(* IEC 61131-3 sources: volt/packages/volt-lsp-iec/test-corpus/bakon-nano/Device/Plc Logic/Application/Library Manager/VisuUtils, 38 files *)

(* ---- CLOSEDIALOGDATA.dut ---- *)
TYPE CLOSEDIALOGDATA :
STRUCT
	DLGMANAGER : VisuElemBase.IDialogManager;
	VISUDIALOG : VisuElemBase.IVisualisationDialog;
	DIALOGRESULT : VisuElemBase.Visu_DialogResult;
END_STRUCT
END_TYPE

(* ---- ERROR.dut ---- *)
TYPE ERROR :
(
	NO_ERROR,
	TIME_OUT,
	NOT_CALLED_FROM_VISU,
	NOT_SUPPORTED_FOR_INTEGRATED_VISU,
	ERROR,
	TRANSFER_CANCELLED,
	TRANSER_IN_PROGRESS,
	TRANSFER_FAILED,
	FILE_READ_ERROR,
	VISU_NOT_FOUND,
	NO_CLIENT_FILTER,
	NO_ITERATION_CALLBACK,
	FILE_TRANSFER_SERVICES_NOT_SUPPORTED,
	BLOCKED_DUE_TO_ONLINECHANGE,
	CANCELLED_DUE_TO_ONLINE_CHANGE
);
END_TYPE

(* ---- OPENDIALOGDATA.dut ---- *)
TYPE OPENDIALOGDATA :
STRUCT
	DLGMANAGER : VisuElemBase.IDialogManager;
	VISUDIALOG : VisuElemBase.IVisualisationDialog;
	POSITIONRECT : VisuElemBase.VisuStructSimpleRectangle;
END_STRUCT
END_TYPE

(* ---- VISUINPUTTYPE.dut ---- *)
TYPE VISUINPUTTYPE :
(
	KEYBOARD := 0,
	TOUCHSCREEN := 1
);
END_TYPE

(* ---- GLOBALS.gvl ---- *)
VAR_GLOBAL
	ALLCLIENTS : FBAcceptsAllClients;
	CURRENTCLIENT : FBAcceptsCurrentClient;
	ONLYTARGETVISU : FBAcceptsTargetVisuOnly;
	ONLYREMOTETARGETVISU : FBAcceptsRemoteTargetVisuOnly;
	ONLYWEBVISU : FBAcceptsWebVisuOnly;
END_VAR

(* ---- PUBLICVARIABLES.gvl ---- *)
VAR_GLOBAL
	CLIENTS : FbCurrentClientProvider;
END_VAR

(* ---- VARIABLES.gvl ---- *)
VAR_GLOBAL
	G_ACTIONHANDLER_INST : FbActionHandler;
	G_OCDETECTOR : FBOCStateDetector;
END_VAR

(* ---- ICAPTURECURRENTCLIENT.itf ---- *)
INTERFACE ICAPTURECURRENTCLIENT
END_INTERFACE

(* ---- IEXECUTEACTION.itf ---- *)
INTERFACE IEXECUTEACTION
END_INTERFACE

METHOD STARTEXECUTE
END_METHOD

(* ---- IVISUALIZATIONCLIENT.itf ---- *)
INTERFACE IVISUALIZATIONCLIENT
END_INTERFACE

METHOD GETCLIENTNAME : STRING
VAR_OUTPUT
	XISVALID : BOOL;
END_VAR
END_METHOD

METHOD GETIPV4ADDRESS : STRING
VAR_OUTPUT
	XISVALID : BOOL;
END_VAR
END_METHOD

METHOD GETREMOTETARGETVISUID : DWORD
VAR_OUTPUT
	XISVALID : BOOL;
END_VAR
END_METHOD

METHOD GETREMOTETARGETVISUVERSION : VERSION
VAR_OUTPUT
	XISVALID : BOOL;
END_VAR
END_METHOD

(* ---- IVISUALIZATIONCLIENTFILTER.itf ---- *)
INTERFACE IVISUALIZATIONCLIENTFILTER
END_INTERFACE

METHOD ISACCEPTED : BOOL
VAR_INPUT
	ITFCLIENT : IVisualizationClient;
END_VAR
END_METHOD

(* ---- IVISUALIZATIONCLIENTITERATION.itf ---- *)
INTERFACE IVISUALIZATIONCLIENTITERATION
END_INTERFACE

METHOD ENDITERATION
END_METHOD

METHOD HANDLECLIENT
VAR_INPUT
	ITFCLIENT : IVisualizationClient;
END_VAR
END_METHOD

METHOD STARTITERATION
END_METHOD

(* ---- IVISUALIZATIONCLIENTRAW.itf ---- *)
INTERFACE IVISUALIZATIONCLIENTRAW
END_INTERFACE

(* ---- FCTGETNEXTVISU.pou ---- *)
FUNCTION FCTGETNEXTVISU : IVisualisation
VAR_INPUT
	PCLIENT : POINTER TO VisuStructClientData;
END_VAR
END_FUNCTION

(* ---- FCTGETPREVIOUSVISU.pou ---- *)
FUNCTION FCTGETPREVIOUSVISU : IVisualisation
VAR_INPUT
	PCLIENT : POINTER TO VisuStructClientData;
END_VAR
END_FUNCTION

(* ---- GETCLIENTTAGIPV4.pou ---- *)
FUNCTION GETCLIENTTAGIPV4 : BOOL
VAR_INPUT
	PCLIENTDATA : POINTER TO VisuStructClientData;
END_VAR
VAR_IN_OUT
	SIPV4 : STRING;
END_VAR
END_FUNCTION

(* ---- GETCLIENTTAGNAME.pou ---- *)
FUNCTION GETCLIENTTAGNAME : BOOL
VAR_INPUT
	PCLIENTDATA : POINTER TO VisuStructClientData;
END_VAR
VAR_IN_OUT
	SNAME : STRING;
END_VAR
END_FUNCTION

(* ---- GETCLIENTTAGREMOTETARGETVISUID.pou ---- *)
FUNCTION GETCLIENTTAGREMOTETARGETVISUID : BOOL
VAR_INPUT
	PCLIENTDATA : POINTER TO VisuStructClientData;
END_VAR
VAR_OUTPUT
	DWID : DWORD;
END_VAR
END_FUNCTION

(* ---- GETCLIENTTAGREMOTETARGETVISUVERSION.pou ---- *)
FUNCTION GETCLIENTTAGREMOTETARGETVISUVERSION : BOOL
VAR_INPUT
	PCLIENTDATA : POINTER TO VisuStructClientData;
END_VAR
VAR_IN_OUT
	V : VERSION;
END_VAR
END_FUNCTION

(* ---- ISVISUTASK.pou ---- *)
FUNCTION ISVISUTASK : BOOL
END_FUNCTION

(* ---- FBACCEPTSALLCLIENTS.pou ---- *)
FUNCTION_BLOCK FBACCEPTSALLCLIENTS
END_FUNCTION_BLOCK

METHOD ISACCEPTED : BOOL
VAR_INPUT
	ITFCLIENT : IVisualizationClient;
END_VAR
END_METHOD

(* ---- FBACCEPTSCLIENTBYTYPEBASE.pou ---- *)
FUNCTION_BLOCK FBACCEPTSCLIENTBYTYPEBASE
VAR
	ABSTRACCEPTEDCLIENTTYPE : VisuClientType;
END_VAR
END_FUNCTION_BLOCK

METHOD ISACCEPTED : BOOL
VAR_INPUT
	ITFCLIENT : IVisualizationClient;
END_VAR
END_METHOD

(* ---- FBACCEPTSCURRENTCLIENT.pou ---- *)
FUNCTION_BLOCK FBACCEPTSCURRENTCLIENT
END_FUNCTION_BLOCK

METHOD ISACCEPTED : BOOL
VAR_INPUT
	ITFCLIENT : IVisualizationClient;
END_VAR
END_METHOD

METHOD SETCLIENT
VAR_INPUT
	PCLIENTDATA : POINTER TO VisuElemBase.VisuStructClientData;
END_VAR
END_METHOD

(* ---- FBACCEPTSREMOTETARGETVISUONLY.pou ---- *)
FUNCTION_BLOCK FBACCEPTSREMOTETARGETVISUONLY EXTENDS FBAcceptsClientByTypeBase
VAR
	ABSTRACCEPTEDCLIENTTYPE : VisuClientType;
END_VAR
END_FUNCTION_BLOCK

(* ---- FBACCEPTSTARGETVISUONLY.pou ---- *)
FUNCTION_BLOCK FBACCEPTSTARGETVISUONLY EXTENDS FBAcceptsClientByTypeBase
VAR
	ABSTRACCEPTEDCLIENTTYPE : VisuClientType;
END_VAR
END_FUNCTION_BLOCK

(* ---- FBACCEPTSWEBVISUONLY.pou ---- *)
FUNCTION_BLOCK FBACCEPTSWEBVISUONLY EXTENDS FBAcceptsClientByTypeBase
VAR
	ABSTRACCEPTEDCLIENTTYPE : VisuClientType;
END_VAR
END_FUNCTION_BLOCK

(* ---- FBACTIONHANDLER.pou ---- *)
FUNCTION_BLOCK FBACTIONHANDLER
VAR
	AACTIONFBINFO : ARRAY [0..(MAX_ACTIONS - 1)] OF IExecuteAction;
	USIFBCOUNT : USINT := 0;
	HSEM : SysSem.RTS_IEC_HANDLE := SysSem.RTS_INVALID_HANDLE;
	MAX_ACTIONS : USINT := 10;
END_VAR
END_FUNCTION_BLOCK

METHOD ADDACTIONFB
VAR_INPUT
	ITFACTIONFBTOADD : IExecuteAction;
END_VAR
END_METHOD

METHOD EXECUTEACTION
END_METHOD

METHOD FB_EXIT : BOOL
VAR_INPUT
	BINCOPYCODE : BOOL;
END_VAR
END_METHOD

METHOD FB_INIT
VAR_INPUT
	BINITRETAINS : BOOL;
	BINCOPYCODE : BOOL;
END_VAR
END_METHOD

METHOD REMOVEACTIONFB : BOOL
VAR_INPUT
	ITFACTIONFBTOREMOVE : IExecuteAction;
END_VAR
END_METHOD

(* ---- FBCHANGEVISU.pou ---- *)
FUNCTION_BLOCK FBCHANGEVISU EXTENDS FbExecuteSingleVisuActionBase
VAR_INPUT
	SVISUNAME : STRING;
END_VAR
END_FUNCTION_BLOCK

METHOD DOEXECUTE
END_METHOD

METHOD DOEXECUTEFORCLIENT
VAR_INPUT
	PCLIENT : POINTER TO VisuElemBase.VisuStructClientData;
	PBYDATA : POINTER TO BYTE;
END_VAR
END_METHOD

(* ---- FBCLIENTWRAPPER.pou ---- *)
FUNCTION_BLOCK FBCLIENTWRAPPER
VAR
	_PCLIENT : POINTER TO VisuStructClientData;
	_ICLIENTID : INT;
	_ECLIENTTYPE : VisuClientType;
	CLIENTDATAPOINTER : POINTER TO VisuElemBase.VisuStructClientData;
	CLIENTDEVICEPIXELRATIO : REAL;
	CLIENTHEIGHT : INT;
	CLIENTID : INT;
	CLIENTTYPE : VisuClientType;
	CLIENTWIDTH : INT;
	CURRENTVISUNAME : STRING;
	INPUTTYPE : VisuInputType;
	NEXTVISUNAME : STRING;
	PREVIOUSVISUNAME : STRING;
	USERGROUPID : DWORD;
	USERNAME : WSTRING;
END_VAR
END_FUNCTION_BLOCK

METHOD GETCLIENTNAME : STRING
VAR_OUTPUT
	XISVALID : BOOL;
END_VAR
END_METHOD

METHOD GETIPV4ADDRESS : STRING
VAR_OUTPUT
	XISVALID : BOOL;
END_VAR
END_METHOD

METHOD GETREMOTETARGETVISUID : DWORD
VAR_OUTPUT
	XISVALID : BOOL;
END_VAR
END_METHOD

METHOD GETREMOTETARGETVISUVERSION : VERSION
VAR_OUTPUT
	XISVALID : BOOL;
END_VAR
END_METHOD

METHOD SETCLIENT
VAR_INPUT
	PCLIENTDATA : POINTER TO VisuElemBase.VisuStructClientData;
END_VAR
END_METHOD

(* ---- FBCLOSEDIALOG.pou ---- *)
FUNCTION_BLOCK FBCLOSEDIALOG EXTENDS FbExecuteSingleVisuActionBase
VAR_INPUT
	SDIALOGNAME : STRING;
	DIALOGRESULT : VisuElemBase.Visu_DialogResult;
END_VAR
VAR
	_SDIALOGNAME : STRING;
	DIALOGFLAGS : DWORD := 0;
END_VAR
END_FUNCTION_BLOCK

METHOD ACTIONDONE
VAR_INPUT
	EACTIONTYPE : VisuElemBase.VisuEnumActionType;
	PCLIENTDATA : POINTER TO VisuElemBase.VisuStructClientData;
END_VAR
END_METHOD

METHOD DOEXECUTE
END_METHOD

METHOD DOEXECUTEFORCLIENT
VAR_INPUT
	PCLIENT : POINTER TO VisuElemBase.VisuStructClientData;
	PBYDATA : POINTER TO BYTE;
END_VAR
END_METHOD

METHOD DOSTARTACTION
END_METHOD

(* ---- FBCURRENTCLIENTPROVIDER.pou ---- *)
FUNCTION_BLOCK FBCURRENTCLIENTPROVIDER
VAR
	CW : FbClientWrapper;
	CURRENT : IVisualizationClient;
END_VAR
END_FUNCTION_BLOCK

(* ---- FBEXECUTESINGLEVISUACTIONBASE.pou ---- *)
FUNCTION_BLOCK FBEXECUTESINGLEVISUACTIONBASE EXTENDS ETrig
VAR_INPUT
	ITFCLIENTFILTER : IVisualizationClientFilter;
END_VAR
VAR_OUTPUT
	EERROR : ERROR;
END_VAR
VAR
	_XACTIONDONE : BOOL := FALSE;
	_PCURRENTCLIENTDATA : POINTER TO VisuStructClientData;
	_IONLINECHANGESTARTVALUE : INT;
END_VAR
END_FUNCTION_BLOCK

METHOD CYCLICACTION
VAR_INPUT
	ITFTIMINGCONTROLLER : CBML.ITimingController;
END_VAR
VAR_OUTPUT
	XCOMPLETE : BOOL;
	IERRORID : INT;
END_VAR
END_METHOD

METHOD FB_EXIT : BOOL
VAR_INPUT
	BINCOPYCODE : BOOL;
END_VAR
END_METHOD

METHOD STARTACTION
VAR_OUTPUT
	XCOMPLETE : BOOL;
	IERRORID : INT;
END_VAR
END_METHOD

METHOD STARTEXECUTE
END_METHOD

METHOD DOEXECUTE
END_METHOD

METHOD DOEXECUTEFORCLIENT
VAR_INPUT
	PCLIENT : POINTER TO VisuElemBase.VisuStructClientData;
	PBYDATA : POINTER TO BYTE;
END_VAR
END_METHOD

METHOD DOSTARTACTION
END_METHOD

METHOD ONCYCLICACTIONDONE : BOOL
VAR_OUTPUT
	XCOMPLETE : BOOL;
	IERRORID : INT;
END_VAR
END_METHOD

METHOD ITERATECLIENTS
VAR_INPUT
	PDATA : POINTER TO BYTE;
END_VAR
END_METHOD

(* ---- FBFILETRANSFER.pou ---- *)
FUNCTION_BLOCK FBFILETRANSFER EXTENDS FbExecuteSingleVisuActionBase
VAR_INPUT
	EDIRECTION : VisuElemBase.VisuEnumFileTransferDirection;
	SPLCFILEPATH : STRING(255);
	SOPTVISUFILEPATH : STRING(255);
END_VAR
VAR
	_XTRANSFERACTIVE : BOOL;
	_XTRANSFERSUCCESSFUL : BOOL;
	_ETRANSFERERROR : VisuElemBase.VisuEnumFileTransferError;
END_VAR
END_FUNCTION_BLOCK

METHOD DOEXECUTE
END_METHOD

METHOD DOEXECUTEFORCLIENT
VAR_INPUT
	PCLIENT : POINTER TO VisuElemBase.VisuStructClientData;
	PBYDATA : POINTER TO BYTE;
END_VAR
END_METHOD

METHOD MAPERROR : ERROR
VAR_INPUT
	ETRANSFERERROR : VisuElemBase.VisuEnumFileTransferError;
END_VAR
END_METHOD

METHOD ONCYCLICACTIONDONE : BOOL
VAR_OUTPUT
	XCOMPLETE : BOOL;
	IERRORID : INT;
END_VAR
END_METHOD

(* ---- FBITERATECLIENTS.pou ---- *)
FUNCTION_BLOCK FBITERATECLIENTS EXTENDS FbExecuteSingleVisuActionBase
VAR_INPUT
	ITFITERATIONCALLBACK : IVisualizationClientIteration;
END_VAR
END_FUNCTION_BLOCK

METHOD STARTACTION
VAR_OUTPUT
	XCOMPLETE : BOOL;
	IERRORID : INT;
END_VAR
END_METHOD

METHOD DOEXECUTE
END_METHOD

METHOD DOEXECUTEFORCLIENT
VAR_INPUT
	PCLIENT : POINTER TO VisuElemBase.VisuStructClientData;
	PBYDATA : POINTER TO BYTE;
END_VAR
END_METHOD

(* ---- FBOCSTATEDETECTOR.pou ---- *)
FUNCTION_BLOCK FBOCSTATEDETECTOR
VAR_OUTPUT
	XDURINGVISUONLINECHANGE : BOOL;
	IOCCOUNTER : INT;
END_VAR
END_FUNCTION_BLOCK

METHOD FB_EXIT : BOOL
VAR_INPUT
	BINCOPYCODE : BOOL;
END_VAR
END_METHOD

METHOD FB_INIT
VAR_INPUT
	BINITRETAINS : BOOL;
	BINCOPYCODE : BOOL;
END_VAR
END_METHOD

(* ---- FBOPENDIALOG.pou ---- *)
FUNCTION_BLOCK FBOPENDIALOG EXTENDS FbExecuteSingleVisuActionBase
VAR_INPUT
	SDIALOGNAME : STRING;
	XMODAL : BOOL := TRUE;
	PTOPLEFTPOSITION : POINTER TO VisuStructPoint;
END_VAR
VAR
	_SDIALOGNAME : STRING;
	DIALOGFLAGS : DWORD := 0;
END_VAR
END_FUNCTION_BLOCK

METHOD ACTIONDONE
VAR_INPUT
	EACTIONTYPE : VisuElemBase.VisuEnumActionType;
	PCLIENTDATA : POINTER TO VisuElemBase.VisuStructClientData;
END_VAR
END_METHOD

METHOD CALLOPENDIALOG
VAR_INPUT
	VISUDIALOG : VisuElemBase.IVisualisationDialog;
	DLGMANAGER : VisuElemBase.IDialogManager;
	PPOSITIONRECT : POINTER TO VisuElemBase.VisuStructSimpleRectangle;
	PCLIENTDATATOUSE : POINTER TO VisuElemBase.VisuStructClientData;
END_VAR
END_METHOD

METHOD DOEXECUTE
END_METHOD

METHOD DOEXECUTEFORCLIENT
VAR_INPUT
	PCLIENT : POINTER TO VisuElemBase.VisuStructClientData;
	PBYDATA : POINTER TO BYTE;
END_VAR
END_METHOD

METHOD DOSTARTACTION
END_METHOD

(* ---- FBOPENDIALOGEXTENDED.pou ---- *)
FUNCTION_BLOCK FBOPENDIALOGEXTENDED EXTENDS FbOpenDialog
VAR_INPUT
	ITFDIALOGOPENEDLISTENER : VisuElemBase.IDialogOpenedListener;
	PBYDIALOGINTERFACEDATA : POINTER TO BYTE;
	UDIDIALOGINTERFACEDATASIZE : UDINT;
	ITFDIALOGCLOSELISTENER : VisuElemBase.IDialogCloseListener;
	PBYTAGFORDIALOGCLOSED : POINTER TO BYTE;
	DWDIALOGFLAGS : DWORD;
END_VAR
VAR
	M_IDSTACKFORELEMENT : VisuElemBase.VisuClientObjectIdStack;
	ITFCAPTURECURRENTCLIENT : ICaptureCurrentClient;
END_VAR
END_FUNCTION_BLOCK

METHOD CALLOPENDIALOG
VAR_INPUT
	VISUDIALOG : VisuElemBase.IVisualisationDialog;
	DLGMANAGER : VisuElemBase.IDialogManager;
	PPOSITIONRECT : POINTER TO VisuElemBase.VisuStructSimpleRectangle;
	PCLIENTDATATOUSE : POINTER TO VisuElemBase.VisuStructClientData;
END_VAR
END_METHOD

(* ---- VISUCLIENTTYPE.dut ---- *)
TYPE VISUCLIENTTYPE :
(
	UNKNOWN := 16#0,
	PROGRAMMINGSYSTEM := 16#1,
	TARGETVISUALIZATION := 16#4,
	WEBVISUALIZATION := 16#8,
	REMOTETARGETVISUALIZATION := 16#10,
	ALLREMOTEVISUALIZATIONS := 16#1B
);
END_TYPE
